(* IEC 61131-3 sources: AXOpen/src/core/ctrl/src/abstractions/IxMessage, 2 files *)

(* ---- IIxMessageCategorize.st ---- *)
NAMESPACE ix.framework.core
    INTERFACE IIxMessageCategorize
		/// <summary>
        /// Categorizes and creates the message as 'debug'.
		/// </summary>
        METHOD AsDebug : IIxMessageProperties END_METHOD

		/// <summary>
        /// Categorizes and creates the message as 'error'.
		/// </summary>
        METHOD AsError : IIxMessageProperties END_METHOD

		/// <summary>
        /// Categorizes and creates the message as 'fatal'.
		/// </summary>
        METHOD AsFatal : IIxMessageProperties END_METHOD

		/// <summary>
        /// Categorizes and creates the message as 'info'.
		/// </summary>
        METHOD AsInfo : IIxMessageProperties END_METHOD

		/// <summary>
        /// Categorizes and creates the message as 'trace'.
		/// </summary>
        METHOD AsTrace : IIxMessageProperties END_METHOD

		/// <summary>
        /// Categorizes and creates the message as 'warning'.
		/// </summary>
        METHOD AsWarning : IIxMessageProperties END_METHOD
    END_INTERFACE
END_NAMESPACE

(* ---- IIxMessageTextBuilder.st ---- *)
NAMESPACE ix.framework.core
    INTERFACE IIxMessageTextBuilder
		/// <summary>
		/// Appends string to the message text.
		/// </summary>
		/// <remarks>
		/// 	<note type="warning">
		/// 		The size of the resulting string should not be more than '160' characters. The characters exceeding this size will be truncated.
		/// 	</note>
		/// </remarks>
        METHOD Append : IIxMessageTextBuilder
            VAR_INPUT
                Text : STRING[IxIntConstants#MAX_MESSAGE_TEXT_LENGHT];
            END_VAR
        END_METHOD

		/// <summary>
		/// Gets categorization methods for fluent message builder.
		/// </summary>
        METHOD As : IIxMessageCategorize END_METHOD

		/// <summary>
		/// Initiates new message text building for this messenger in fluent-like fashion.
		/// </summary>
        METHOD Build : IIxMessageTextBuilder END_METHOD
    END_INTERFACE
END_NAMESPACE
